FUNCTION_BLOCK FB_DataSim
VAR_INPUT
END_VAR
VAR_OUTPUT
	rValue: REAL := 1.0000;
END_VAR
VAR
	CountTimer: TON;
	RisingEdge: R_TRIG;
	DataStack: FB_Messwerte;
END_VAR

CountTimer(IN := TRUE, PT := T#2S);
RisingEdge(CLK:= CountTimer.Q);

IF RisingEdge.Q AND rValue < 10000 THEN
	rValue := rValue * LREAL_TO_REAL(PI);
	DataStack(rValue := rValue);
ELSIF RisingEdge.Q AND rValue > 10000 THEN
	rValue := (rValue /100) * 1.75;
	DataStack(rValue := rValue);
END_IF

IF CountTimer.Q THEN
	CountTimer(IN := FALSE);
	CountTimer(IN := TRUE);
END_IF

END_FUNCTION_BLOCK

(* stored: Version 1.1.0.1
   POU FB_DataSim: Id {74b0651b-ac84-4077-a6ac-bb2adacc5a02}, SpecialFunc None *)
